Universal Robots PolyScope program: test1218.urp

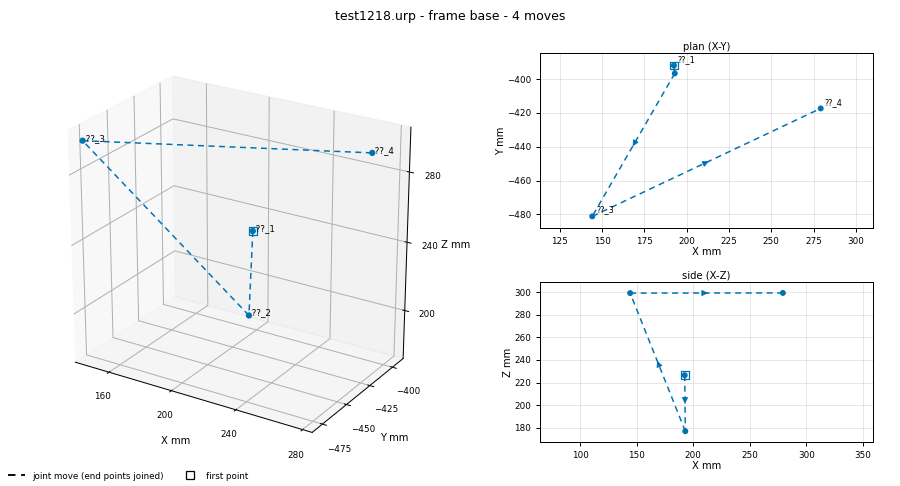
[picture p0: tool path of test1218.urp in frame base, 4 of 4 moves have a stored position in this frame; points joined in program order, loops and branches not executed]
Program test1218 (installation=20240827 directory=/programs createdIn=5.15.1 lastSavedIn=5.15.1 robotSerialNumber=20245500285)
Calibrated DH parameters: a=[0.000097, -0.210459, -0.026602, 0.000137, 0.000078, 0]; d=[0.162601, 254.180657, -54.076236, -199.970743, 0.099615, 0.099684]; alpha=[1.569796, -0.001455, 0.001957, 1.570525, -1.571561, 0]; deltaTheta=[0, -1.053331, 8.839472, -1.50296, 0.000002, 0]
InitVariablesNode
Robot Program (runOnlyOnce=false)
  MoveJ speed 60 deg/s, acceleration 80 deg/s^2 (useActiveTCP=true) feature=Base
    Waypoint 路点_1: TCP in base x=192.487 y=-391.985 z=226.496 mm, rx=1.9742 ry=2.4231 rz=0.1108 rad; joints [95.805, -98.902, 107.766, -96.613, -86.544, 84.238] deg; TCP offset x=-0.17 y=0 z=192.95 mm, rx=0 ry=0 rz=0 rad
    Waypoint 路点_2: TCP in base x=192.979 y=-396.627 z=176.976 mm, rx=-1.9378 ry=-2.37 rz=-0.239 rad; joints [95.804, -92.021, 107.764, -96.606, -86.548, 84.235] deg
    Waypoint 路点_3: TCP in base x=144.202 y=-481.152 z=299.134 mm, rx=-2.1598 ry=-2.2472 rz=0.1006 rad; joints [93.339, -91.462, 91.372, -91.484, -93.595, 91.183] deg
    Waypoint 路点_4: TCP in base x=279.272 y=-417.335 z=299.267 mm, rx=-1.8073 ry=-2.5518 rz=0.1054 rad; joints [110.435, -91.5, 91.395, -91.495, -93.584, 91.167] deg
